(*
SPDX-FileCopyrightText: © 2026 Oleksandr Tiutyk <trofimich@gmail.com>
SPDX-License-Identifier: MIT
License: https://opensource.org/license/mit
*)

(*!
<summary>Exposes diagnostics for failed explicit initialization.</summary>
<description>
Uses the GeneralException lifetime and throw rules. The initialization diagnostic is copied from a
WSTRING(255) input.
</description>
*)
INTERFACE IClassInitializationException EXTENDS IGeneralException

(*!
<summary>Reports failed initialization of the specified class.</summary>
<description>
Combines the class name with the diagnostic text and raises the exception. The errorMessage input is copied by
value and limited to 255 characters.
</description>
*)
METHOD Throw
VAR_INPUT
	sourceNamespaceName : STRING;
	sourceClassName : STRING;
	sourcePOUName : STRING;
	sourcePosition : STRING;
	errorMessage : WSTRING(255);
END_VAR
END_METHOD

END_INTERFACE

(* stored: Version 1.1.0.1
   Itf IClassInitializationException: Id {42616ec1-02de-435c-bf47-8aeec77b916f}
   Method Throw: Id {b133f255-3d05-44fb-b413-a6a39115e0f3} *)
